Universal Robots PolyScope program: IAC007 Sensors B.urp

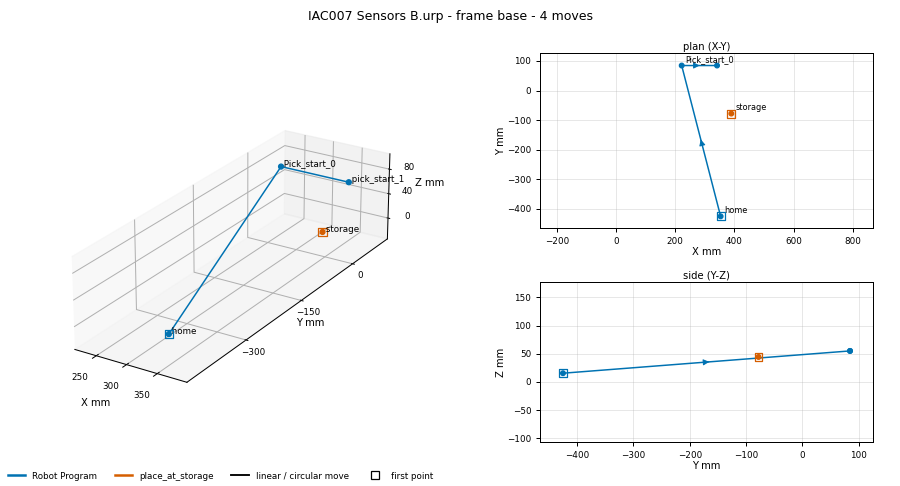
[picture p0: tool path of IAC007 Sensors B.urp in frame base, 4 of 5 moves have a stored position in this frame; points joined in program order, loops and branches not executed]
Program IAC007 Sensors B (installation=default directory=/programs createdIn=5.9.1.1031110 lastSavedIn=5.9.1.1031110 robotSerialNumber=20195501059)
Calibrated DH parameters: a=[0.000146, -0.418764, -0.053981, 0.000058, -0.000023, 0]; d=[0.162545, 37.319448, -206.067439, 168.881546, 0.09955, 0.099464]; alpha=[1.57004, -0.001979, 0.002304, 1.570607, -1.57066, 0]; deltaTheta=[0, -0.174616, -1.258233, 1.432844, -0.000001, 0]
BeforeStart
  URCap Gripper Activate (Robotiq_Grippers, Robotiq Inc.) dataModel(ResetAndActivateKey=false)
  initial_p := get_actual_tcp_pose()
  MoveJ speed 60 deg/s, acceleration 80 deg/s^2 (useActiveTCP=true) feature=Base
    Waypoint Waypoint (Variable): variable=initial_p
Robot Program (runOnlyOnce=true)
  URCap Grip Check (Robotiq_Grippers, Robotiq Inc.) dataModel(ObjectDetectedKey=true, DimensionValidationKey=false, DimensionKey=100.0, DimensionDimensionPositiveGapKey=5.0, DimensionNegativeGapKey=5.0, GripperIdKey=1, ModelDefinedKey=true); state(isChildrenLocked=true)
    URCap If (Robotiq_Grippers, Robotiq Inc.)
      Popup Error (haltProgram=false message=Object in gripper. Safe to open? inputType=Text)
      URCap Gripper (Robotiq_Grippers, Robotiq Inc.) dataModel(position=0.0, force=1.0, speed=20.0, positionInDouble=0.0, forceInDouble=1.0, speedInDouble=20.0, slaveIds=[9], blocking=true)
  MoveL speed 250 mm/s, acceleration 1200 mm/s^2 (useActiveTCP=true) feature=Base
    MoveDirectionNode (selectedDirection=ZMinus) feature=Joint_6_name
      Until DISTANCE (allowActions=false deceleration=3 distanceNodeType=STOP) Distance=0.05; motionParameters(blendRadius=0)
  URCap Gripper (Robotiq_Grippers, Robotiq Inc.) dataModel(position=100.0, force=100.0, speed=100.0, positionInDouble=100.0, forceInDouble=100.0, speedInDouble=100.0, slaveIds=[9], blocking=true)
  MoveL speed 250 mm/s, acceleration 1200 mm/s^2 (useActiveTCP=true) feature=Base
    Waypoint home: TCP in base x=353.442 y=-425.051 z=15.364 mm, rx=-2.1827 ry=-2.2594 rz=0 rad; joints [115.734, -68.978, 112.532, -133.544, 270.037, 113.795] deg; TCP offset x=0 y=0 z=174 mm, rx=0 ry=0 rz=0 rad
  Loop Forever
    URCap Grip Check (Robotiq_Grippers, Robotiq Inc.) dataModel(DimensionKey=100.0, DimensionDimensionPositiveGapKey=5.0, DimensionNegativeGapKey=5.0, GripperIdKey=1, ModelDefinedKey=true, ObjectDetectedKey=false, DimensionValidationKey=false); state(isChildrenLocked=true)
      URCap If (Robotiq_Grippers, Robotiq Inc.)
        If not digital_in[0]
          MoveL speed 250 mm/s, acceleration 1200 mm/s^2 (useActiveTCP=true) feature=Base
            Waypoint Pick_start_0: TCP in base x=221.928 y=84.351 z=54.912 mm, rx=2.1827 ry=2.2595 rz=-0.0001 rad; joints [166.668, -126.792, 153.163, -116.361, 270.111, 164.668] deg
            Call pick
            Call place_at_storage
        If not digital_in[1]
          MoveL speed 250 mm/s, acceleration 1200 mm/s^2 (useActiveTCP=true) feature=Base
            Waypoint pick_start_1: TCP in base x=341.369 y=84.377 z=54.889 mm, rx=-2.1827 ry=-2.2594 rz=0.0001 rad; joints [171.568, -100.099, 140.138, -130.026, 270.095, 169.618] deg
            Call pick
            Call place_at_storage
SubProgram -> pick
SubProgram -> place_at_storage
SubProgram pick (keepSynchronizedWithDisk=false)
  URCap Gripper (Robotiq_Grippers, Robotiq Inc.) dataModel(position=100.0, force=100.0, speed=100.0, positionInDouble=100.0, forceInDouble=100.0, speedInDouble=100.0, slaveIds=[9], blocking=true)
  MoveL speed 250 mm/s, acceleration 1200 mm/s^2 (useActiveTCP=true) feature=Base
    MoveDirectionNode (selectedDirection=ZPlus toolParams=0.02, 0.5) feature=Joint_6_name
      Until TOOL_CONTACT_DETECTION (allowActions=true retraction=0.002 decelerationAcceleration=3 decelerationAngularAcceleration=34.906585)
        URCap Gripper (Robotiq_Grippers, Robotiq Inc.) dataModel(position=0.0, force=100.0, speed=100.0, positionInDouble=0.0, forceInDouble=100.0, speedInDouble=100.0, slaveIds=[9], blocking=true)
        MoveDirectionNode (selectedDirection=ZPlus toolParams=0.02, 0.5) feature=Joint_6_name
          Until TOOL_CONTACT_DETECTION (allowActions=false retraction=0.002 decelerationAcceleration=3 decelerationAngularAcceleration=34.906585)
        URCap Gripper (Robotiq_Grippers, Robotiq Inc.) dataModel(position=100.0, force=1.0, speed=20.0, positionInDouble=100.0, forceInDouble=1.0, speedInDouble=20.0, slaveIds=[9], blocking=true)
        MoveDirectionNode (selectedDirection=ZPlus) feature=Base
          Until DISTANCE (allowActions=false deceleration=3 distanceNodeType=STOP) Distance=0.035; motionParameters(blendRadius=0)
      Until DISTANCE (allowActions=true deceleration=3 distanceNodeType=STOP) Distance=0.025; motionParameters(blendRadius=0)
        Popup Error (haltProgram=false message=object not found inputType=Text)
SubProgram place_at_storage (keepSynchronizedWithDisk=false)
  MoveL speed 250 mm/s, acceleration 1200 mm/s^2 (useActiveTCP=true) feature=Base
    Waypoint storage: TCP in base x=389.556 y=-77.98 z=44.175 mm, rx=-2.1825 ry=-2.2597 rz=0.0001 rad; joints [149.031, -91.397, 134.803, -133.396, 270.08, 147.079] deg
    MoveDirectionNode (selectedDirection=ZPlus toolParams=0.02, 0.5) feature=Joint_6_name
      Until TOOL_CONTACT_DETECTION (allowActions=false retraction=0 decelerationAcceleration=3 decelerationAngularAcceleration=34.906585)
    URCap Gripper (Robotiq_Grippers, Robotiq Inc.) dataModel(position=0.0, force=1.0, speed=20.0, positionInDouble=0.0, forceInDouble=1.0, speedInDouble=20.0, slaveIds=[9], blocking=true)
    MoveDirectionNode (selectedDirection=ZPlus)
      Until DISTANCE (allowActions=false deceleration=3 distanceNodeType=STOP) Distance=0.05; motionParameters(blendRadius=0)
